// TIA Portal V19 export
TYPE "Positioning_DOL_Machine_CIn"
// stored: Access Published
   STRUCT
      Manager : "Positioning_DOL_Machine_Manager";
      MinusExtEnable : Bool;
      PlusExtEnable : Bool;
      ExternalPowerOn : Bool;
      ExternalAlarms : Bool;
      PositionLimits : Struct
         EnableMin : Bool;
         PosMin : LReal;
         EnableMax : Bool;
         PosMax : LReal;
      END_STRUCT;
   END_STRUCT;
END_TYPE
